(* CODESYS project STAS-60.project

Project tree, tasks and I/O mapping:
  Device : XC303 (Preview), Eaton Automation, version 3.5.11.10
      unmapped channels: Output, Input
    application Application
      libraries: Standard, * (System); CAA CiA 405, 3.5.8.0 (CAA Technical Workgroup); Serial Communication, 3.5.7.0 (3S - Smart Software Solutions GmbH)
      task MainTask (cyclic, interval t#200ms, priority 1) calls PLC_PRG
      task VISU_TASK (cyclic, interval t#200ms, priority 1) calls VisuElems.Visu_Prg
      task TrendRecordingTask (cyclic, interval 100 ms, priority 31) calls VisuTrendStorageAccess.GlobalInstances.g_TrendRecordingManager.CyclicCall
      program PLC_PRG [ST]
      global variables GVL
      visualisation Visualization
    CANbus : CANbus, Eaton Automation, order no. 
      , version 3.5.10.0
      CANopen_Manager : CANopen_Manager, Eaton Automation, order no. 
      , version 3.5.10.0
          settings: ConfigVersion = 50659584
        XNE_GWBR_CANOPEN : XNE-GWBR-CANOPEN, Eaton Automation, order no. 107591, version Revision=16#00040017, FileVersion=4.24
            settings: NODEIDSAVED = 2; SDO Timeout = 1000000; PDO_Autoconfig = TRUE; EXPERTSETTINGS = False; Emergency-General Parameters.Emergency COBID = 16#00000082; Heartbeat-Producer Time = 200; Settings.COBID = 16#00000202; Settings.Transmission Type = 16#FF; Settings.available PDO-Parameter.Inhibit Time available = FALSE; Settings.available PDO-Parameter.Event Timer available = FALSE; Settings.Inhibit Time = 0; Settings.Event Timer = 0; Generic COBID = '$NODEID+16#0200'; Process by CANopenManager = TRUE; Settings.COBID = 16#00000302; Settings.Transmission Type = 16#FF; Settings.available PDO-Parameter.Inhibit Time available = FALSE; Settings.available PDO-Parameter.Event Timer available = FALSE; Settings.Inhibit Time = 0; Settings.Event Timer = 0; Generic COBID = '$NODEID+16#0300'; Process by CANopenManager = TRUE; Settings.COBID = 16#00000282; Settings.Transmission Type = 16#FF; Settings.available PDO-Parameter.Inhibit Time available = TRUE; Settings.available PDO-Parameter.Event Timer available = TRUE; Settings.Inhibit Time = 0; Settings.Event Timer = 0; Generic COBID = '$NODEID+16#0280'; Process by CANopenManager = TRUE; Settings.COBID = 16#00000382; Settings.Transmission Type = 16#FF; Settings.available PDO-Parameter.Inhibit Time available = TRUE; Settings.available PDO-Parameter.Event Timer available = TRUE; Settings.Inhibit Time = 0; Settings.Event Timer = 0; Generic COBID = '$NODEID+16#0380'; Process by CANopenManager = TRUE; Heartbeat-Consuming1.Heartbeat-Time = 300 ms; WriteOutput8Bit : Generic_XN_2DO.Index = 16#6200;
              WriteOutput8Bit : Generic_XN_2DO.Subindex = 16#01; WriteOutput8Bit : Generic_XN_2DO.ObjectLength = 8; WriteOutput8Bit : Generic_XN_2DO_4.Index = 16#6200; WriteOutput8Bit : Generic_XN_2DO_4.Subindex = 16#02; WriteOutput8Bit : Generic_XN_2DO_4.ObjectLength = 8; WriteAnalogueOutput16 : Generic_XNE_4AO.Index = 16#6411; WriteAnalogueOutput16 : Generic_XNE_4AO.Subindex = 16#01; WriteAnalogueOutput16 : Generic_XNE_4AO.ObjectLength = 16; WriteAnalogueOutput16 : Generic_XNE_4AO.Index = 16#6411; WriteAnalogueOutput16 : Generic_XNE_4AO.Subindex = 16#02; WriteAnalogueOutput16 : Generic_XNE_4AO.ObjectLength = 16; WriteAnalogueOutput16 : Generic_XNE_4AO.Index = 16#6411; WriteAnalogueOutput16 : Generic_XNE_4AO.Subindex = 16#03; WriteAnalogueOutput16 : Generic_XNE_4AO.ObjectLength = 16; WriteAnalogueOutput16 : Generic_XNE_4AO.Index = 16#6411; WriteAnalogueOutput16 : Generic_XNE_4AO.Subindex = 16#04; WriteAnalogueOutput16 : Generic_XNE_4AO.ObjectLength = 16; ReadAnalogueInput16Bit : Generic_XNE_8AI.Index = 16#6401; ReadAnalogueInput16Bit : Generic_XNE_8AI.Subindex = 16#01; ReadAnalogueInput16Bit : Generic_XNE_8AI.ObjectLength = 16; ReadAnalogueInput16Bit : Generic_XNE_8AI.Index = 16#6401; ReadAnalogueInput16Bit : Generic_XNE_8AI.Subindex = 16#02; ReadAnalogueInput16Bit : Generic_XNE_8AI.ObjectLength = 16; ReadAnalogueInput16Bit : Generic_XNE_8AI.Index = 16#6401; ReadAnalogueInput16Bit : Generic_XNE_8AI.Subindex = 16#03; ReadAnalogueInput16Bit : Generic_XNE_8AI.ObjectLength = 16; ReadAnalogueInput16Bit : Generic_XNE_8AI.Index = 16#6401; ReadAnalogueInput16Bit : Generic_XNE_8AI.Subindex = 16#04; ReadAnalogueInput16Bit : Generic_XNE_8AI.ObjectLength = 16; ReadAnalogueInput16Bit : Generic_XNE_8AI.Index = 16#6401; ReadAnalogueInput16Bit : Generic_XNE_8AI.Subindex = 16#05; ReadAnalogueInput16Bit : Generic_XNE_8AI.ObjectLength = 16; ReadAnalogueInput16Bit : Generic_XNE_8AI.Index = 16#6401; ReadAnalogueInput16Bit : Generic_XNE_8AI.Subindex = 16#06; ReadAnalogueInput16Bit : Generic_XNE_8AI.ObjectLength = 16; ReadAnalogueInput16Bit : Generic_XNE_8AI.Index = 16#6401; ReadAnalogueInput16Bit : Generic_XNE_8AI.Subindex = 16#07; ReadAnalogueInput16Bit : Generic_XNE_8AI.ObjectLength = 16; ReadAnalogueInput16Bit : Generic_XNE_8AI.Index = 16#6401; ReadAnalogueInput16Bit : Generic_XNE_8AI.Subindex = 16#08;
              ReadAnalogueInput16Bit : Generic_XNE_8AI.ObjectLength = 16; SDO List.Set Guardtime.Index = 16#100C; SDO List.Set Guardtime.Subindex = 16#00; SDO List.Set Guardtime.Value = 16#00000000; SDO List.Set Guardtime.Size = 16; SDO List.Set Guardtime.AbortIfError = FALSE; SDO List.Set Guardtime.JumpToLine = FALSE; SDO List.Set Guardtime.Line = 0; SDO List.Set Lifetime.Index = 16#100D; SDO List.Set Lifetime.Subindex = 16#00; SDO List.Set Lifetime.Value = 16#00000000; SDO List.Set Lifetime.Size = 8; SDO List.Set Lifetime.AbortIfError = FALSE; SDO List.Set Lifetime.JumpToLine = FALSE; SDO List.Set Lifetime.Line = 0; SDO List.Disable Emcy CobID.Index = 16#1014; SDO List.Disable Emcy CobID.Subindex = 16#00; SDO List.Disable Emcy CobID.Value = 16#80000082; SDO List.Disable Emcy CobID.Size = 32; SDO List.Disable Emcy CobID.AbortIfError = FALSE; SDO List.Disable Emcy CobID.JumpToLine = FALSE; SDO List.Disable Emcy CobID.Line = 0; SDO List.Set Emcy CobID.Index = 16#1014; SDO List.Set Emcy CobID.Subindex = 16#00; SDO List.Set Emcy CobID.Value = 16#00000082; SDO List.Set Emcy CobID.Size = 32; SDO List.Set Emcy CobID.AbortIfError = FALSE; SDO List.Set Emcy CobID.JumpToLine = FALSE; SDO List.Set Emcy CobID.Line = 0; SDO List.Set Heartbeat Consumer.Index = 16#1016; SDO List.Set Heartbeat Consumer.Subindex = 16#01; SDO List.Set Heartbeat Consumer.Value = 16#0001012C; SDO List.Set Heartbeat Consumer.Size = 32; SDO List.Set Heartbeat Consumer.AbortIfError = FALSE; SDO List.Set Heartbeat Consumer.JumpToLine = FALSE; SDO List.Set Heartbeat Consumer.Line = 0; SDO List.Set Heartbeat Producer.Index = 16#1017; SDO List.Set Heartbeat Producer.Subindex = 16#00; SDO List.Set Heartbeat Producer.Value = 16#000000C8; SDO List.Set Heartbeat Producer.Size = 16;
              SDO List.Set Heartbeat Producer.AbortIfError = FALSE; SDO List.Set Heartbeat Producer.JumpToLine = FALSE; SDO List.Set Heartbeat Producer.Line = 0; SDO List.Disable PDO.Index = 16#1400; SDO List.Disable PDO.Subindex = 16#01; SDO List.Disable PDO.Value = 16#80000202; SDO List.Disable PDO.Size = 32; SDO List.Disable PDO.AbortIfError = FALSE; SDO List.Disable PDO.JumpToLine = FALSE; SDO List.Disable PDO.Line = 0; SDO List.Set transmission type.Index = 16#1400; SDO List.Set transmission type.Subindex = 16#02; SDO List.Set transmission type.Value = 16#FF; SDO List.Set transmission type.Size = 8; SDO List.Set transmission type.AbortIfError = FALSE; SDO List.Set transmission type.JumpToLine = FALSE; SDO List.Set transmission type.Line = 0; SDO List.Clear pdo mapping.Index = 16#1600; SDO List.Clear pdo mapping.Subindex = 16#00; SDO List.Clear pdo mapping.Value = 16#0; SDO List.Clear pdo mapping.Size = 8; SDO List.Clear pdo mapping.AbortIfError = FALSE; SDO List.Clear pdo mapping.JumpToLine = FALSE; SDO List.Clear pdo mapping.Line = 0; SDO List.Set Mapping.Index = 16#1600; SDO List.Set Mapping.Subindex = 16#01; SDO List.Set Mapping.Value = 16#62000108; SDO List.Set Mapping.Size = 32; SDO List.Set Mapping.AbortIfError = FALSE; SDO List.Set Mapping.JumpToLine = FALSE; SDO List.Set Mapping.Line = 0; SDO List.Set Mapping.Index = 16#1600; SDO List.Set Mapping.Subindex = 16#02; SDO List.Set Mapping.Value = 16#62000208; SDO List.Set Mapping.Size = 32; SDO List.Set Mapping.AbortIfError = FALSE; SDO List.Set Mapping.JumpToLine = FALSE; SDO List.Set Mapping.Line = 0; SDO List.Set number of mappings.Index = 16#1600; SDO List.Set number of mappings.Subindex = 16#00;
              SDO List.Set number of mappings.Value = 16#02; SDO List.Set number of mappings.Size = 8; SDO List.Set number of mappings.AbortIfError = FALSE; SDO List.Set number of mappings.JumpToLine = FALSE; SDO List.Set number of mappings.Line = 0; SDO List.Set and enable COB-ID.Index = 16#1400; SDO List.Set and enable COB-ID.Subindex = 16#01; SDO List.Set and enable COB-ID.Value = 16#00000202; SDO List.Set and enable COB-ID.Size = 32; SDO List.Set and enable COB-ID.AbortIfError = FALSE; SDO List.Set and enable COB-ID.JumpToLine = FALSE; SDO List.Set and enable COB-ID.Line = 0; SDO List.Disable PDO.Index = 16#1401; SDO List.Disable PDO.Subindex = 16#01; SDO List.Disable PDO.Value = 16#80000302; SDO List.Disable PDO.Size = 32; SDO List.Disable PDO.AbortIfError = FALSE; SDO List.Disable PDO.JumpToLine = FALSE; SDO List.Disable PDO.Line = 0; SDO List.Set transmission type.Index = 16#1401; SDO List.Set transmission type.Subindex = 16#02; SDO List.Set transmission type.Value = 16#FF; SDO List.Set transmission type.Size = 8; SDO List.Set transmission type.AbortIfError = FALSE; SDO List.Set transmission type.JumpToLine = FALSE; SDO List.Set transmission type.Line = 0; SDO List.Clear pdo mapping.Index = 16#1601; SDO List.Clear pdo mapping.Subindex = 16#00; SDO List.Clear pdo mapping.Value = 16#0; SDO List.Clear pdo mapping.Size = 8; SDO List.Clear pdo mapping.AbortIfError = FALSE; SDO List.Clear pdo mapping.JumpToLine = FALSE; SDO List.Clear pdo mapping.Line = 0; SDO List.Set Mapping.Index = 16#1601; SDO List.Set Mapping.Subindex = 16#01; SDO List.Set Mapping.Value = 16#64110110; SDO List.Set Mapping.Size = 32; SDO List.Set Mapping.AbortIfError = FALSE; SDO List.Set Mapping.JumpToLine = FALSE; SDO List.Set Mapping.Line = 0;
              SDO List.Set Mapping.Index = 16#1601; SDO List.Set Mapping.Subindex = 16#02; SDO List.Set Mapping.Value = 16#64110210; SDO List.Set Mapping.Size = 32; SDO List.Set Mapping.AbortIfError = FALSE; SDO List.Set Mapping.JumpToLine = FALSE; SDO List.Set Mapping.Line = 0; SDO List.Set Mapping.Index = 16#1601; SDO List.Set Mapping.Subindex = 16#03; SDO List.Set Mapping.Value = 16#64110310; SDO List.Set Mapping.Size = 32; SDO List.Set Mapping.AbortIfError = FALSE; SDO List.Set Mapping.JumpToLine = FALSE; SDO List.Set Mapping.Line = 0; SDO List.Set Mapping.Index = 16#1601; SDO List.Set Mapping.Subindex = 16#04; SDO List.Set Mapping.Value = 16#64110410; SDO List.Set Mapping.Size = 32; SDO List.Set Mapping.AbortIfError = FALSE; SDO List.Set Mapping.JumpToLine = FALSE; SDO List.Set Mapping.Line = 0; SDO List.Set number of mappings.Index = 16#1601; SDO List.Set number of mappings.Subindex = 16#00; SDO List.Set number of mappings.Value = 16#04; SDO List.Set number of mappings.Size = 8; SDO List.Set number of mappings.AbortIfError = FALSE; SDO List.Set number of mappings.JumpToLine = FALSE; SDO List.Set number of mappings.Line = 0; SDO List.Set and enable COB-ID.Index = 16#1401; SDO List.Set and enable COB-ID.Subindex = 16#01; SDO List.Set and enable COB-ID.Value = 16#00000302; SDO List.Set and enable COB-ID.Size = 32; SDO List.Set and enable COB-ID.AbortIfError = FALSE; SDO List.Set and enable COB-ID.JumpToLine = FALSE; SDO List.Set and enable COB-ID.Line = 0; SDO List.Disable PDO.Index = 16#1801; SDO List.Disable PDO.Subindex = 16#01; SDO List.Disable PDO.Value = 16#80000282; SDO List.Disable PDO.Size = 32; SDO List.Disable PDO.AbortIfError = FALSE;
              SDO List.Disable PDO.JumpToLine = FALSE; SDO List.Disable PDO.Line = 0; SDO List.Set transmission type.Index = 16#1801; SDO List.Set transmission type.Subindex = 16#02; SDO List.Set transmission type.Value = 16#FF; SDO List.Set transmission type.Size = 8; SDO List.Set transmission type.AbortIfError = FALSE; SDO List.Set transmission type.JumpToLine = FALSE; SDO List.Set transmission type.Line = 0; SDO List.Set inhibit time.Index = 16#1801; SDO List.Set inhibit time.Subindex = 16#03; SDO List.Set inhibit time.Value = 16#0000; SDO List.Set inhibit time.Size = 16; SDO List.Set inhibit time.AbortIfError = FALSE; SDO List.Set inhibit time.JumpToLine = FALSE; SDO List.Set inhibit time.Line = 0; SDO List.Set event time.Index = 16#1801; SDO List.Set event time.Subindex = 16#05; SDO List.Set event time.Value = 16#0000; SDO List.Set event time.Size = 16; SDO List.Set event time.AbortIfError = FALSE; SDO List.Set event time.JumpToLine = FALSE; SDO List.Set event time.Line = 0; SDO List.Clear pdo mapping.Index = 16#1A01; SDO List.Clear pdo mapping.Subindex = 16#00; SDO List.Clear pdo mapping.Value = 16#0; SDO List.Clear pdo mapping.Size = 8; SDO List.Clear pdo mapping.AbortIfError = FALSE; SDO List.Clear pdo mapping.JumpToLine = FALSE; SDO List.Clear pdo mapping.Line = 0; SDO List.Set Mapping.Index = 16#1A01; SDO List.Set Mapping.Subindex = 16#01; SDO List.Set Mapping.Value = 16#64010110; SDO List.Set Mapping.Size = 32; SDO List.Set Mapping.AbortIfError = FALSE; SDO List.Set Mapping.JumpToLine = FALSE; SDO List.Set Mapping.Line = 0; SDO List.Set Mapping.Index = 16#1A01; SDO List.Set Mapping.Subindex = 16#02; SDO List.Set Mapping.Value = 16#64010210;
              SDO List.Set Mapping.Size = 32; SDO List.Set Mapping.AbortIfError = FALSE; SDO List.Set Mapping.JumpToLine = FALSE; SDO List.Set Mapping.Line = 0; SDO List.Set Mapping.Index = 16#1A01; SDO List.Set Mapping.Subindex = 16#03; SDO List.Set Mapping.Value = 16#64010310; SDO List.Set Mapping.Size = 32; SDO List.Set Mapping.AbortIfError = FALSE; SDO List.Set Mapping.JumpToLine = FALSE; SDO List.Set Mapping.Line = 0; SDO List.Set Mapping.Index = 16#1A01; SDO List.Set Mapping.Subindex = 16#04; SDO List.Set Mapping.Value = 16#64010410; SDO List.Set Mapping.Size = 32; SDO List.Set Mapping.AbortIfError = FALSE; SDO List.Set Mapping.JumpToLine = FALSE; SDO List.Set Mapping.Line = 0; SDO List.Set number of mappings.Index = 16#1A01; SDO List.Set number of mappings.Subindex = 16#00; SDO List.Set number of mappings.Value = 16#04; SDO List.Set number of mappings.Size = 8; SDO List.Set number of mappings.AbortIfError = FALSE; SDO List.Set number of mappings.JumpToLine = FALSE; SDO List.Set number of mappings.Line = 0; SDO List.Set and enable COB-ID.Index = 16#1801; SDO List.Set and enable COB-ID.Subindex = 16#01; SDO List.Set and enable COB-ID.Value = 16#00000282; SDO List.Set and enable COB-ID.Size = 32; SDO List.Set and enable COB-ID.AbortIfError = FALSE; SDO List.Set and enable COB-ID.JumpToLine = FALSE; SDO List.Set and enable COB-ID.Line = 0; SDO List.Disable PDO.Index = 16#1802; SDO List.Disable PDO.Subindex = 16#01; SDO List.Disable PDO.Value = 16#80000382; SDO List.Disable PDO.Size = 32; SDO List.Disable PDO.AbortIfError = FALSE; SDO List.Disable PDO.JumpToLine = FALSE; SDO List.Disable PDO.Line = 0; SDO List.Set transmission type.Index = 16#1802;
              SDO List.Set transmission type.Subindex = 16#02; SDO List.Set transmission type.Value = 16#FF; SDO List.Set transmission type.Size = 8; SDO List.Set transmission type.AbortIfError = FALSE; SDO List.Set transmission type.JumpToLine = FALSE; SDO List.Set transmission type.Line = 0; SDO List.Set inhibit time.Index = 16#1802; SDO List.Set inhibit time.Subindex = 16#03; SDO List.Set inhibit time.Value = 16#0000; SDO List.Set inhibit time.Size = 16; SDO List.Set inhibit time.AbortIfError = FALSE; SDO List.Set inhibit time.JumpToLine = FALSE; SDO List.Set inhibit time.Line = 0; SDO List.Set event time.Index = 16#1802; SDO List.Set event time.Subindex = 16#05; SDO List.Set event time.Value = 16#0000; SDO List.Set event time.Size = 16; SDO List.Set event time.AbortIfError = FALSE; SDO List.Set event time.JumpToLine = FALSE; SDO List.Set event time.Line = 0; SDO List.Clear pdo mapping.Index = 16#1A02; SDO List.Clear pdo mapping.Subindex = 16#00; SDO List.Clear pdo mapping.Value = 16#0; SDO List.Clear pdo mapping.Size = 8; SDO List.Clear pdo mapping.AbortIfError = FALSE; SDO List.Clear pdo mapping.JumpToLine = FALSE; SDO List.Clear pdo mapping.Line = 0; SDO List.Set Mapping.Index = 16#1A02; SDO List.Set Mapping.Subindex = 16#01; SDO List.Set Mapping.Value = 16#64010510; SDO List.Set Mapping.Size = 32; SDO List.Set Mapping.AbortIfError = FALSE; SDO List.Set Mapping.JumpToLine = FALSE; SDO List.Set Mapping.Line = 0; SDO List.Set Mapping.Index = 16#1A02; SDO List.Set Mapping.Subindex = 16#02; SDO List.Set Mapping.Value = 16#64010610; SDO List.Set Mapping.Size = 32; SDO List.Set Mapping.AbortIfError = FALSE; SDO List.Set Mapping.JumpToLine = FALSE;
              SDO List.Set Mapping.Line = 0; SDO List.Set Mapping.Index = 16#1A02; SDO List.Set Mapping.Subindex = 16#03; SDO List.Set Mapping.Value = 16#64010710; SDO List.Set Mapping.Size = 32; SDO List.Set Mapping.AbortIfError = FALSE; SDO List.Set Mapping.JumpToLine = FALSE; SDO List.Set Mapping.Line = 0; SDO List.Set Mapping.Index = 16#1A02; SDO List.Set Mapping.Subindex = 16#04; SDO List.Set Mapping.Value = 16#64010810; SDO List.Set Mapping.Size = 32; SDO List.Set Mapping.AbortIfError = FALSE; SDO List.Set Mapping.JumpToLine = FALSE; SDO List.Set Mapping.Line = 0; SDO List.Set number of mappings.Index = 16#1A02; SDO List.Set number of mappings.Subindex = 16#00; SDO List.Set number of mappings.Value = 16#04; SDO List.Set number of mappings.Size = 8; SDO List.Set number of mappings.AbortIfError = FALSE; SDO List.Set number of mappings.JumpToLine = FALSE; SDO List.Set number of mappings.Line = 0; SDO List.Set and enable COB-ID.Index = 16#1802; SDO List.Set and enable COB-ID.Subindex = 16#01; SDO List.Set and enable COB-ID.Value = 16#00000382; SDO List.Set and enable COB-ID.Size = 32; SDO List.Set and enable COB-ID.AbortIfError = FALSE; SDO List.Set and enable COB-ID.JumpToLine = FALSE; SDO List.Set and enable COB-ID.Line = 0; ConfigVersion = 50659584
          Generic_XN_2DO : Generic XN-2DO, Eaton Automation, order no. 0, version Revision=16#00040017, FileVersion=4.24
              settings: Number of Params = 1; WriteOutput8Bit : Generic_XN_2DO.Index = 16#6200; WriteOutput8Bit : Generic_XN_2DO.Subindex = 16#01; WriteOutput8Bit : Generic_XN_2DO.Startbit = 0; WriteOutput8Bit : Generic_XN_2DO.Endbit = 1
              unmapped channels: WriteOutput8Bit : Generic_XN_2DO
          Generic_XN_2DO_1 : Generic XN-2DO, Eaton Automation, order no. 0, version Revision=16#00040017, FileVersion=4.24
              settings: Number of Params = 1; WriteOutput8Bit : Generic_XN_2DO.Index = 16#6200; WriteOutput8Bit : Generic_XN_2DO.Subindex = 16#01; WriteOutput8Bit : Generic_XN_2DO.Startbit = 2; WriteOutput8Bit : Generic_XN_2DO.Endbit = 3
              unmapped channels: WriteOutput8Bit : Generic_XN_2DO
          Generic_XN_2DO_2 : Generic XN-2DO, Eaton Automation, order no. 0, version Revision=16#00040017, FileVersion=4.24
              settings: Number of Params = 1; WriteOutput8Bit : Generic_XN_2DO.Index = 16#6200; WriteOutput8Bit : Generic_XN_2DO.Subindex = 16#01; WriteOutput8Bit : Generic_XN_2DO.Startbit = 4; WriteOutput8Bit : Generic_XN_2DO.Endbit = 5
              unmapped channels: WriteOutput8Bit : Generic_XN_2DO
          Generic_XN_2DO_3 : Generic XN-2DO, Eaton Automation, order no. 0, version Revision=16#00040017, FileVersion=4.24
              settings: Number of Params = 1; WriteOutput8Bit : Generic_XN_2DO.Index = 16#6200; WriteOutput8Bit : Generic_XN_2DO.Subindex = 16#01; WriteOutput8Bit : Generic_XN_2DO.Startbit = 6; WriteOutput8Bit : Generic_XN_2DO.Endbit = 7
              unmapped channels: WriteOutput8Bit : Generic_XN_2DO
          Generic_XN_2DO_4 : Generic XN-2DO, Eaton Automation, order no. 0, version Revision=16#00040017, FileVersion=4.24
              settings: Number of Params = 1; WriteOutput8Bit : Generic_XN_2DO_4.Index = 16#6200; WriteOutput8Bit : Generic_XN_2DO_4.Subindex = 16#02; WriteOutput8Bit : Generic_XN_2DO_4.Startbit = 0; WriteOutput8Bit : Generic_XN_2DO_4.Endbit = 1
              unmapped channels: WriteOutput8Bit : Generic_XN_2DO_4
          Generic_XN_2DO_5 : Generic XN-2DO, Eaton Automation, order no. 0, version Revision=16#00040017, FileVersion=4.24
              settings: Number of Params = 1; WriteOutput8Bit : Generic_XN_2DO_4.Index = 16#6200; WriteOutput8Bit : Generic_XN_2DO_4.Subindex = 16#02; WriteOutput8Bit : Generic_XN_2DO_4.Startbit = 2; WriteOutput8Bit : Generic_XN_2DO_4.Endbit = 3
              unmapped channels: WriteOutput8Bit : Generic_XN_2DO_4
          Generic_XN_2DO_6 : Generic XN-2DO, Eaton Automation, order no. 0, version Revision=16#00040017, FileVersion=4.24
              settings: Number of Params = 1; WriteOutput8Bit : Generic_XN_2DO_4.Index = 16#6200; WriteOutput8Bit : Generic_XN_2DO_4.Subindex = 16#02; WriteOutput8Bit : Generic_XN_2DO_4.Startbit = 4; WriteOutput8Bit : Generic_XN_2DO_4.Endbit = 5
              unmapped channels: WriteOutput8Bit : Generic_XN_2DO_4
          Generic_XN_2DO_7 : Generic XN-2DO, Eaton Automation, order no. 0, version Revision=16#00040017, FileVersion=4.24
              settings: Number of Params = 1; WriteOutput8Bit : Generic_XN_2DO_4.Index = 16#6200; WriteOutput8Bit : Generic_XN_2DO_4.Subindex = 16#02; WriteOutput8Bit : Generic_XN_2DO_4.Startbit = 6; WriteOutput8Bit : Generic_XN_2DO_4.Endbit = 7
              unmapped channels: WriteOutput8Bit : Generic_XN_2DO_4
          Generic_XNE_4AO : Generic XNE-4AO, Eaton Automation, order no. 0, version Revision=16#00040017, FileVersion=4.24
              settings: Number of Params = 4; WriteAnalogueOutput16 : Generic_XNE_4AO.Index = 16#6411; WriteAnalogueOutput16 : Generic_XNE_4AO.Subindex = 16#01; WriteAnalogueOutput16 : Generic_XNE_4AO.Startbit = 0; WriteAnalogueOutput16 : Generic_XNE_4AO.Endbit = 15; WriteAnalogueOutput16 : Generic_XNE_4AO.Index = 16#6411; WriteAnalogueOutput16 : Generic_XNE_4AO.Subindex = 16#02; WriteAnalogueOutput16 : Generic_XNE_4AO.Startbit = 0; WriteAnalogueOutput16 : Generic_XNE_4AO.Endbit = 15; WriteAnalogueOutput16 : Generic_XNE_4AO.Index = 16#6411; WriteAnalogueOutput16 : Generic_XNE_4AO.Subindex = 16#03; WriteAnalogueOutput16 : Generic_XNE_4AO.Startbit = 0; WriteAnalogueOutput16 : Generic_XNE_4AO.Endbit = 15; WriteAnalogueOutput16 : Generic_XNE_4AO.Index = 16#6411; WriteAnalogueOutput16 : Generic_XNE_4AO.Subindex = 16#04; WriteAnalogueOutput16 : Generic_XNE_4AO.Startbit = 0; WriteAnalogueOutput16 : Generic_XNE_4AO.Endbit = 15
              unmapped channels: WriteAnalogueOutput16 : Generic_XNE_4AO, WriteAnalogueOutput16 : Generic_XNE_4AO, WriteAnalogueOutput16 : Generic_XNE_4AO, WriteAnalogueOutput16 : Generic_XNE_4AO
          Generic_XNE_8AI : Generic XNE-8AI, Eaton Automation, order no. 0, version Revision=16#00040017, FileVersion=4.24
              settings: Number of Params = 8; ReadAnalogueInput16Bit : Generic_XNE_8AI.Index = 16#6401; ReadAnalogueInput16Bit : Generic_XNE_8AI.Subindex = 16#01; ReadAnalogueInput16Bit : Generic_XNE_8AI.Startbit = 0; ReadAnalogueInput16Bit : Generic_XNE_8AI.Endbit = 15; ReadAnalogueInput16Bit : Generic_XNE_8AI.Index = 16#6401; ReadAnalogueInput16Bit : Generic_XNE_8AI.Subindex = 16#02; ReadAnalogueInput16Bit : Generic_XNE_8AI.Startbit = 0; ReadAnalogueInput16Bit : Generic_XNE_8AI.Endbit = 15; ReadAnalogueInput16Bit : Generic_XNE_8AI.Index = 16#6401; ReadAnalogueInput16Bit : Generic_XNE_8AI.Subindex = 16#03; ReadAnalogueInput16Bit : Generic_XNE_8AI.Startbit = 0; ReadAnalogueInput16Bit : Generic_XNE_8AI.Endbit = 15; ReadAnalogueInput16Bit : Generic_XNE_8AI.Index = 16#6401; ReadAnalogueInput16Bit : Generic_XNE_8AI.Subindex = 16#04; ReadAnalogueInput16Bit : Generic_XNE_8AI.Startbit = 0; ReadAnalogueInput16Bit : Generic_XNE_8AI.Endbit = 15; ReadAnalogueInput16Bit : Generic_XNE_8AI.Index = 16#6401; ReadAnalogueInput16Bit : Generic_XNE_8AI.Subindex = 16#05; ReadAnalogueInput16Bit : Generic_XNE_8AI.Startbit = 0; ReadAnalogueInput16Bit : Generic_XNE_8AI.Endbit = 15; ReadAnalogueInput16Bit : Generic_XNE_8AI.Index = 16#6401; ReadAnalogueInput16Bit : Generic_XNE_8AI.Subindex = 16#06; ReadAnalogueInput16Bit : Generic_XNE_8AI.Startbit = 0; ReadAnalogueInput16Bit : Generic_XNE_8AI.Endbit = 15; ReadAnalogueInput16Bit : Generic_XNE_8AI.Index = 16#6401; ReadAnalogueInput16Bit : Generic_XNE_8AI.Subindex = 16#07; ReadAnalogueInput16Bit : Generic_XNE_8AI.Startbit = 0; ReadAnalogueInput16Bit : Generic_XNE_8AI.Endbit = 15; ReadAnalogueInput16Bit : Generic_XNE_8AI.Index = 16#6401; ReadAnalogueInput16Bit : Generic_XNE_8AI.Subindex = 16#08; ReadAnalogueInput16Bit : Generic_XNE_8AI.Startbit = 0; ReadAnalogueInput16Bit : Generic_XNE_8AI.Endbit = 15
              unmapped channels: ReadAnalogueInput16Bit : Generic_XNE_8AI, ReadAnalogueInput16Bit : Generic_XNE_8AI, ReadAnalogueInput16Bit : Generic_XNE_8AI, ReadAnalogueInput16Bit : Generic_XNE_8AI, ReadAnalogueInput16Bit : Generic_XNE_8AI, ReadAnalogueInput16Bit : Generic_XNE_8AI, ReadAnalogueInput16Bit : Generic_XNE_8AI, ReadAnalogueInput16Bit : Generic_XNE_8AI
    Ethernet : Ethernet, Eaton Automation, version 3.5.11.0
      ModbusTCP_Slave_Device : ModbusTCP Slave Device, 3S - Smart Software Solutions GmbH, version 3.5.11.0
          unmapped channels: Входы, Выходы
  libraries: VisuSymbols, 3.5.10.0 (System)
  text list GlobalTextList
*)

// Device/Application/GVL
{attribute 'qualified_only'}
VAR_GLOBAL
	
	hiPres AT %IW2: WORD; (*Датчик высокго давления на гидроразпределителе*)
	lowPres AT %IW4: WORD; (*Датчик низкого давления на гидроразпределителе*)
	mowAbsorb AT %IW6: WORD; (*Датчик хода гидроамортизатора*)
	compressPress AT %IW8: WORD; (*Датчик давления на сжатие*)
	decomressPress AT %IW10: WORD; (*Датчик давления на росжатие*)
	
	temperatuteOil : WORD; (*Датчик температуры масла*)
	levelOil : WORD; (*Датчик уровня масла*)
	
	defectHiPresSens: BOOL; (*Неисправность датчика высокго давления на гидроразпределителе*)
	defectLowPresSens: BOOL; (*Неисправность датчика низкого давления на гидроразпределителе*)
	defectMowAbsorbSens: BOOL; (*Неисправность датчика хода гидроамортизатора*)
	defectDecomressPressSens: BOOL; (*Неисправность датчика давления на росжатие*)
	defectCompressPressSens: BOOL; (*Неисправность датчика давления на сжатие*)
	defectTemperatuteOilSens: BOOL; (*Неисправность датчика температуры масла*)
	defectLevelOilSens: BOOL; (*Неисправность датчика уровня масла*)
		
	SOL1 : BOOL; (* Соленоид высокого давления *)
	SOL2 : BOOL; (* Соленоид низкого давления *)
	SOL3: BOOL; (* Соленоид растяжения *)
	SOL4: BOOL; (* Соленоид сжатия *)
	SOL5: BOOL; (* Соленоид без давления *)
	
	SOL10: BOOL; (* Соленоид перепад давления Сжатие *)
	SOL11: BOOL; (* Соленоид перепад давления Растяжение *)
	
	pumpOn: BOOL; (*Включение насоса*)
	pumpStart: BOOL; (*Разгон насоса*)
	pumpWork: BOOL; (*Рабочий режим насоса*)
	
	timePumpStart: TIME; (*Время разгона насоса*)
	
	heaterOil: BOOL; (*Подогрева масла*)
	coolerOil: BOOL; (*Охлаждение масла*)
	
	
	normalLoadMode: BOOL; (*Режим нормальной нагрузки*)
	openMode: BOOL;  (*Проверка открытия клапана*)
	resistanceMode: BOOL; (*Режим испытания сопротивления ГА без нагрузки (холостой ход)*)
	speedCloseMode: BOOL; (*Скорость закрытия*)
	
	nProcess: INT;
	kokoetoChislo: WORD;

END_VAR

// Device/Application/PLC_PRG
PROGRAM PLC_PRG
VAR

	hiPres : WORD:=10; (*Датчик высокго давления на гидроразпределителе*)
	lowPres : WORD:=10; (*Датчик низкого давления на гидроразпределителе*)
	mowAbsorb : WORD:=10; (*Датчик хода гидроамортизатора*)
	compressPress : WORD:=10; (*Датчик давления на сжатие*)
	decomressPress : WORD:=10; (*Датчик давления на росжатие*)
	
	temperatuteOil : WORD:=10; (*Датчик температуры масла*)
	levelOil : WORD:=10; (*Датчик уровня масла*)
	
	leftMowAbsorb: WORD;
	rightMowAbsorb: WORD;
	
	TONInst : TON ;
	setSOL10: BOOL;
	
	
	TOFInst : TOF;
	timeSOL10: TIME:=T#5S; 
		
	TONPump : TON ;
	setPump: BOOL;
	timePump: TIME:=T#5S;
	
	TONnormalMode:TON;
	TOFnormalMode:TOF;
	setNormalMode: BOOL;
	timeNormalMode : TIME:=T#10S;
	
	countNormalMode : INT:=1;
	
	tonSOL1 : TON;
	tofSOL1 : TOF;
	
	tonSOL2 : TON;
	tofSOL2 : TOF;
	
	tonSOL3 : TON;
	tofSOL3 : TOF;
	
	tonSOL4 : TON;
	tofSOL4 : TOF;
	
	tonSOL10 : TON;
	tofSOL10 : TOF;
	
	tonSOL11 : TON;
	tofSOL11 : TOF;
	
	onButton:BOOL;
	
END_VAR

(*Проверка работоспособности датчиков. Анализ токовой петли*)

onButton:= NOT(GVL.pumpWork);

(*Датчик высокого давления*)
IF (hiPres<4 OR hiPres>20 )THEN
		GVL.defectHiPresSens := TRUE;
		ELSE
		GVL.defectHiPresSens := FALSE;
END_IF

(*Датчик низкого давления*)
IF (lowPres<4 OR lowPres>20 )THEN
		GVL.defectLowPresSens := TRUE;
		ELSE
		GVL.defectLowPresSens := FALSE;
END_IF

(*Датчик сжатия*)
IF (compressPress<4 OR compressPress>20 )THEN
		GVL.defectCompressPressSens := TRUE;
		ELSE
		GVL.defectCompressPressSens := FALSE;
END_IF

(*Датчик расжатия*)
IF (decomressPress<4 OR decomressPress>20 )THEN
		GVL.defectDecomressPressSens := TRUE;
		ELSE
		GVL.defectDecomressPressSens := FALSE;
END_IF

(*Датчик температуры масла*)
IF (temperatuteOil<4 OR temperatuteOil>20 )THEN
		GVL.defectTemperatuteOilSens := TRUE;
		ELSE
		GVL.defectTemperatuteOilSens := FALSE;
END_IF

(*Датчик хода гидроамортизатора*)
IF (mowAbsorb<4 OR mowAbsorb>20 )THEN
		GVL.defectMowAbsorbSens := TRUE;
		ELSE
		GVL.defectMowAbsorbSens := FALSE;
END_IF
(*-----------------------------------------------------------*)

(*Ржеим нагрева и охлаждения масла*)

(*Охлаждение*)
IF (temperatuteOil>=16 AND temperatuteOil<=20) THEN
	GVL.coolerOil:=TRUE;
ELSE
	GVL.coolerOil:=FALSE;
END_IF

(*Нагрев*)
IF (temperatuteOil>=4 AND temperatuteOil<=8) THEN
	GVL.heaterOil:=TRUE;
	//TONInst(IN:= GVL.heaterOil, PT:= timeSOL10, Q=> GVL.SOL10);
	//TOFInst(IN:= GVL.heaterOil, PT:= timeSOL10);						
ELSE
	GVL.heaterOil:=FALSE;	
	//TOFInst(IN:= GVL.heaterOil, PT:= timeSOL10, Q=> GVL.SOL10);
	//TONInst(IN := GVL.heaterOil, PT:= timeSOL10);
END_IF
(*-----------------------------------------------------------*)

(*РАбота с електро насосом *)
IF (GVL.pumpOn = TRUE) THEN	
	IF (GVL.pumpWork = FALSE)THEN
		GVL.pumpStart := TRUE;
		TONPump(IN:=GVL.pumpStart, PT:= timePump,Q=>GVL.pumpWork );
	END_IF
ELSE
	GVL.pumpStart := FALSE;
	GVL.pumpWork := FALSE;
	TONPump(IN:=GVL.pumpStart, PT:= timePump);
END_IF
(*------------------------------------------------------------*)


(*Режим нормальной нагрузки*)
IF (GVL.normalLoadMode = TRUE AND GVL.pumpOn=TRUE) THEN
	
CASE countNormalMode OF
1:
	GVL.SOL1:=TRUE;
	tonSOL10 (IN:=TRUE,PT:=T#3S, Q=>GVL.SOL10);
	tonSOL3 (IN:=TRUE,PT:=T#5S, Q=>GVL.SOL3);
	TONnormalMode (IN:=TRUE,PT:=T#10S, Q=>GVL.SOL5);
	
	IF (GVL.SOL5=TRUE) THEN
		TONnormalMode (IN:=FALSE,PT:=T#0S);
		TOFnormalMode (IN:=TRUE,PT:=T#0S);
		tonSOL10 (IN:=FALSE,PT:=T#0S);
		tonSOL3 (IN:=FALSE,PT:=T#0S);
		countNormalMode:=2;
	END_IF
2:
	TOFnormalMode (IN:=FALSE,PT:=T#3S, Q=>GVL.SOL5);
	IF (GVL.SOL5=FALSE) THEN
		TOFnormalMode (IN:=TRUE,PT:=T#0S);		
		countNormalMode:=3;
	END_IF

3:
	tofSOL10 (IN:=FALSE,PT:=T#4S, Q=>GVL.SOL10);
	tofSOL3 (IN:=FALSE,PT:=T#2S, Q=>GVL.SOL3);
	IF (GVL.SOL10=FALSE) THEN
		tofSOL10 (IN:=TRUE,PT:=T#0S);
		tofSOL3 (IN:=TRUE,PT:=T#0S);
	countNormalMode:=4;
	END_IF
4:
	tonSOL11 (IN:=TRUE,PT:=T#3S, Q=>GVL.SOL11);
	tonSOL4 (IN:=TRUE,PT:=T#6S, Q=>GVL.SOL4);
	TONnormalMode (IN:=TRUE,PT:=T#10S, Q=>GVL.SOL5);
	IF (GVL.SOL5=TRUE) THEN
		TONnormalMode (IN:=FALSE,PT:=T#0S);
		tonSOL11 (IN:=FALSE,PT:=T#0S);
		tonSOL4 (IN:=FALSE,PT:=T#0S);
		countNormalMode:=5;
	END_IF
	
5:
	TOFnormalMode (IN:=FALSE,PT:=T#2S, Q=>GVL.SOL5);
	IF (GVL.SOL5=FALSE) THEN
		TOFnormalMode (IN:=TRUE,PT:=T#0S);		
		countNormalMode:=6;
	END_IF
	
6:
	tofSOL11 (IN:=FALSE,PT:=T#4S, Q=>GVL.SOL11);
	tofSOL4 (IN:=FALSE,PT:=T#2S, Q=>GVL.SOL4);
	IF (GVL.SOL11=FALSE) THEN
		tofSOL11 (IN:=TRUE,PT:=T#0S);
		tofSOL4 (IN:=TRUE,PT:=T#0S);
	countNormalMode:=7;
	END_IF
ELSE
	
	countNormalMode:=1;
	GVL.normalLoadMode := FALSE;
		GVL.SOL1:=FALSE;
END_CASE;

END_IF
(*-------------------------------------------------------------*)

(*Режим проверки открытия клапанов*)
IF (GVL.openMode = TRUE AND GVL.pumpOn=TRUE) THEN
	CASE countNormalMode OF	
	1:
		GVL.SOL1:=TRUE;
		tonSOL10 (IN:=TRUE,PT:=T#3S, Q=>GVL.SOL10);
		tonSOL3 (IN:=TRUE,PT:=T#5S, Q=>GVL.SOL3);
		TONnormalMode (IN:=TRUE,PT:=T#10S, Q=>GVL.SOL5);
	
		IF (mowAbsorb>=24) THEN
			TONnormalMode (IN:=FALSE,PT:=T#0S);
			TOFnormalMode (IN:=TRUE,PT:=T#0S);
			tonSOL10 (IN:=FALSE,PT:=T#0S);
			tonSOL3 (IN:=FALSE,PT:=T#0S);
			countNormalMode:=2;
		END_IF
	
	2:
		TOFnormalMode (IN:=FALSE,PT:=T#3S, Q=>GVL.SOL5);
		IF (GVL.SOL5=FALSE) THEN
			TOFnormalMode (IN:=TRUE,PT:=T#0S);		
			countNormalMode:=3;
		END_IF
	
	3:
		tofSOL10 (IN:=FALSE,PT:=T#4S, Q=>GVL.SOL10);
		tofSOL3 (IN:=FALSE,PT:=T#2S, Q=>GVL.SOL3);
		IF (GVL.SOL10=FALSE) THEN
		tofSOL10 (IN:=TRUE,PT:=T#0S);
		tofSOL3 (IN:=TRUE,PT:=T#0S);
		countNormalMode:=4;
		END_IF
	
	4:
		tonSOL11 (IN:=TRUE,PT:=T#3S, Q=>GVL.SOL11);
		tonSOL4 (IN:=TRUE,PT:=T#6S, Q=>GVL.SOL4);
		TONnormalMode (IN:=TRUE,PT:=T#10S, Q=>GVL.SOL5);
		IF (mowAbsorb<=14) THEN
		TONnormalMode (IN:=FALSE,PT:=T#0S);
		tonSOL11 (IN:=FALSE,PT:=T#0S);
		tonSOL4 (IN:=FALSE,PT:=T#0S);
		countNormalMode:=5;
		END_IF
	
	5:
		TOFnormalMode (IN:=FALSE,PT:=T#2S, Q=>GVL.SOL5);
		IF (GVL.SOL5=FALSE) THEN
		TOFnormalMode (IN:=TRUE,PT:=T#0S);		
		countNormalMode:=6;
		END_IF
	
	6:
		tofSOL11 (IN:=FALSE,PT:=T#4S, Q=>GVL.SOL11);
		tofSOL4 (IN:=FALSE,PT:=T#2S, Q=>GVL.SOL4);
		IF (GVL.SOL11=FALSE) THEN
		tofSOL11 (IN:=TRUE,PT:=T#0S);
		tofSOL4 (IN:=TRUE,PT:=T#0S);
		countNormalMode:=7;
		END_IF
	
	ELSE
		countNormalMode:=1;
		GVL.openMode := FALSE;
		GVL.SOL1:=FALSE;
	END_CASE
END_IF
(*-------------------------------------------------------------*)

(*Испытание на сопротивление ГА без нагрузки*)
IF (GVL.resistanceMode = TRUE AND GVL.pumpOn=TRUE) THEN
	
CASE countNormalMode OF
	1:
		GVL.SOL2:=TRUE;
		//tonSOL10 (IN:=TRUE,PT:=T#3S, Q=>GVL.SOL10);
		tonSOL3 (IN:=TRUE,PT:=T#5S, Q=>GVL.SOL3);
		TONnormalMode (IN:=TRUE,PT:=T#10S, Q=>GVL.SOL5);
				
		IF (mowAbsorb>=29) THEN
			TONnormalMode (IN:=FALSE,PT:=T#0S);
			TOFnormalMode (IN:=TRUE,PT:=T#0S);
			//tonSOL10 (IN:=FALSE,PT:=T#0S);
			tonSOL3 (IN:=FALSE,PT:=T#0S);
			countNormalMode:=2;
		END_IF
	2:
		TOFnormalMode (IN:=FALSE,PT:=T#3S, Q=>GVL.SOL5);
		IF (GVL.SOL5=FALSE) THEN
			TOFnormalMode (IN:=TRUE,PT:=T#0S);		
			countNormalMode:=3;
		END_IF
		
	3:
		//tofSOL10 (IN:=FALSE,PT:=T#4S, Q=>GVL.SOL10);
		tofSOL3 (IN:=FALSE,PT:=T#2S, Q=>GVL.SOL3);
		IF (GVL.SOL3=FALSE) THEN
		//tofSOL10 (IN:=TRUE,PT:=T#0S);
		tofSOL3 (IN:=TRUE,PT:=T#0S);
		countNormalMode:=4;
		END_IF
	
	4:
		//tonSOL11 (IN:=TRUE,PT:=T#3S, Q=>GVL.SOL11);
		tonSOL4 (IN:=TRUE,PT:=T#6S, Q=>GVL.SOL4);
		TONnormalMode (IN:=TRUE,PT:=T#10S, Q=>GVL.SOL5);
		IF (mowAbsorb<=9) THEN
		TONnormalMode (IN:=FALSE,PT:=T#0S);
		//tonSOL11 (IN:=FALSE,PT:=T#0S);
		tonSOL4 (IN:=FALSE,PT:=T#0S);
		countNormalMode:=5;
		END_IF
	
	5:
		TOFnormalMode (IN:=FALSE,PT:=T#2S, Q=>GVL.SOL5);
		IF (GVL.SOL5=FALSE) THEN
		TOFnormalMode (IN:=TRUE,PT:=T#0S);		
		countNormalMode:=6;
		END_IF
		
	6:
		//tofSOL11 (IN:=FALSE,PT:=T#4S, Q=>GVL.SOL11);
		tofSOL4 (IN:=FALSE,PT:=T#2S, Q=>GVL.SOL4);
		IF (GVL.SOL4=FALSE) THEN
		//tofSOL11 (IN:=TRUE,PT:=T#0S);
		tofSOL4 (IN:=TRUE,PT:=T#0S);
		countNormalMode:=7;
		END_IF
		
	ELSE
		countNormalMode:=1;
		GVL.resistanceMode := FALSE;
		GVL.SOL2:=FALSE;
	
END_CASE

END_IF
(*-------------------------------------------------------------*)

(*Испытание скорости закрытия клапанов ГА*)
(*-------------------------------------------------------------*)

IF (mowAbsorb>=19 AND mowAbsorb<34) THEN	
rightMowAbsorb:=mowAbsorb-19;
END_IF

IF (mowAbsorb>4 AND mowAbsorb<=19) THEN	
leftMowAbsorb:=19-mowAbsorb;
END_IF

END_PROGRAM

// Device/Application/Visualization
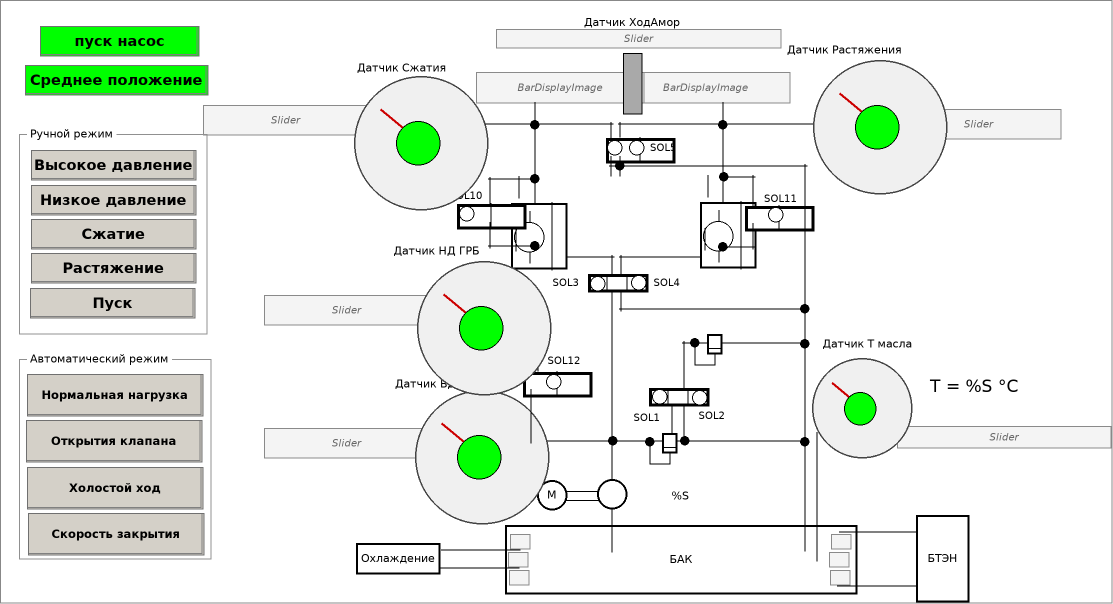
VISUALIZATION Visualization  // 1113x604
VAR_IN_OUT
END_VAR
VAR
	bResetTrigger : BOOL;
	bStop : BOOL;
	bStore : BOOL;
	sStoreFilename : STRING;
	bRestore : BOOL;
	sRestoreFilename : STRING;
END_VAR
    Rectangle (505,525 352x69), "БАК"
    Line (684,443) (684,341), colour toggle: GVL.SOL2
    Line (805,441) (505,441), colour toggle: GVL.pumpWork
    Line (805,343) (682,343), colour toggle: GVL.SOL2
    Slider (897,426 214x22), variable: PLC_PRG.temperatuteOil, scale 0..24
    Rectangle (927,371 95x30), "T = %S °C", text variable: PLC_PRG.temperatuteOil
    Slider (264,428 165x30), variable: PLC_PRG.hiPres, scale 0..25
    Slider (264,295 165x30), variable: PLC_PRG.lowPres, scale 0..25
    Slider (203,105 165x30), variable: PLC_PRG.compressPress, scale 0..25
    Slider (896,109 165x30), variable: PLC_PRG.decomressPress, scale 0..25
    Label (388,236 97x30), "Датчик НД ГРБ"
    Label (389,369 97x30), "Датчик ВД ГРБ"
    Label (353,53 97x30), "Датчик Сжатия"
    Label (779,35 131x30), "Датчик Растяжения"
    Slider (496,29 285x19), variable: PLC_PRG.mowAbsorb, scale 0..36
    BarDisplayImage (621,72 169x31), value: PLC_PRG.rightMowAbsorb, style: BarDisplayImage-Gray, scale format: %.1f, scale 0..15
    BarDisplayImage (476,72 168x31), value: PLC_PRG.leftMowAbsorb, style: BarDisplayImage-Gray, scale format: %.1f, scale 0..15
    Rectangle (623,53 19x61), colour toggle: GVL.defectMowAbsorbSens
    Label (582,13 100x19), "Датчик ХодАмор"
    Line (554,110)
    Ellipse (615,161 9x9)
    Line (603,215)
    Line (613,124) (534,124)
    Line (721,124) (618,124)
    Ellipse (530,120 9x9)
    Ellipse (718,120 9x9)
    Group (606,137 40x19)
        Rectangle (0,1 69x25)
        Line (34,24) (34,0)
    Label (647,138 33x19), "SOL5"
    Line (611,138) (611,122)
    Line (620,137) (620,122)
    Line (723,259) (723,124), colour toggle: GVL.SOL4
    Line (725,257) (619,257), colour toggle: GVL.SOL4
    Line (535,259) (535,124), colour toggle: GVL.SOL3
    Line (614,257) (533,257), colour toggle: GVL.SOL3
    Group (700,175 32x59)
        Rectangle (0,27 56x66)
        Ellipse (3,46 30x30)
        Line (41,94) (41,26)
        Line (8,22) (8,0)
        Line (5,75) (5,53)
        Line (19,46) (19,35)
        Line (19,87) (19,76)
    Group (745,205 40x19)
        Rectangle (0,1 69x25)
        Line (34,24) (34,0)
    Label (763,189 35x19), "SOL11"
    Line (755,177) (722,177), colour toggle: GVL.SOL11
    Line (755,247) (722,247), colour toggle: GVL.SOL11
    Line (753,206) (753,175), colour toggle: GVL.SOL11
    Line (753,249) (753,223), colour toggle: GVL.SOL11
    Ellipse (719,172 9x9)
    Ellipse (718,242 9x9)
    Group (511,176 32x59)
        Rectangle (0,27 56x66)
        Ellipse (3,46 30x30)
        Line (41,94) (41,26)
        Line (8,22) (8,0)
        Line (5,75) (5,53)
        Line (19,46) (19,35)
        Line (19,87) (19,76)
    Group (457,203 40x19)
        Rectangle (0,1 69x25)
        Line (34,24) (34,0)
    Label (448,186 36x19), "SOL10"
    Line (536,179) (488,179), colour toggle: GVL.SOL10
    Line (537,246) (488,246), colour toggle: GVL.SOL10
    Line (490,248) (490,222), colour toggle: GVL.SOL10
    Line (490,205) (490,177), colour toggle: GVL.SOL10
    Group (588,274 60x18)
        Rectangle (0,0 60x18)
        Line (39,17) (39,0)
        Line (19,17) (19,0)
    Line (621,311) (621,291)
    Line (612,552) (612,291), colour toggle: GVL.pumpWork
    Line (621,275) (621,255), colour toggle: GVL.SOL4
    Line (612,275) (612,255), colour toggle: GVL.SOL3
    Line (805,309) (619,309)
    Label (649,273 36x19), "SOL4"
    Label (548,273 36x19), "SOL3"
    Group (692,334 30x41)
        Rectangle (15,0 15x20)
        Line (15,14) (29,14)
        Line (0,40)
        Line (23,31) (23,20)
        Line (23,31) (3,31)
        Line (3,31) (3,8)
    Group (649,388 60x18)
        Rectangle (0,0 60x18)
        Line (39,17) (39,0)
        Line (19,17) (19,0)
    Group (647,433 30x41)
        Rectangle (15,0 15x20)
        Line (15,14) (29,14)
        Line (0,40)
        Line (23,31) (23,20)
        Line (23,31) (3,31)
        Line (3,31) (3,8)
    Line (672,433) (672,406), colour toggle: GVL.SOL1
    Ellipse (530,174 9x9)
    Ellipse (530,241 9x9)
    Ellipse (690,338 9x9)
    Ellipse (645,437 9x9)
    Ellipse (680,436 9x9)
    Group (611,156 10x12)
        Line (9,20) (9,0)
        Line (0,20) (0,0)
    Line (807,166) (609,166)
    Ellipse (597,479 30x30), colour toggle: GVL.pumpWork
    Ellipse (537,480 30x30), "M", colour toggle: GVL.pumpStart
    Line (566,491) (598,491)
    Line (566,500) (598,500)
    Line (805,551) (805,164)
    Ellipse (800,304 9x9)
    Ellipse (800,339 9x9)
    Ellipse (800,437 9x9)
    Ellipse (608,436 9x9)
    Pie (830,570 20x15), colour toggle: GVL.heaterOil
    Line (918,532) (839,532), colour toggle: GVL.heaterOil
    Line (916,586) (837,586), colour toggle: GVL.heaterOil
    Rectangle (916,515 53x87), "БТЭН", colour toggle: GVL.heaterOil
    Group (413,390 100x100)
        Meter360 (0,0 138x134), value: PLC_PRG.hiPres, style: Meter-Meter360-Gray, scale format: %.1f, scale 4..20
        Ellipse (44,45 44x44), colour toggle: GVL.defectHiPresSens
    Line (534,124) (445,124), colour toggle: GVL.SOL3
    Group (352,76 100x100)
        Meter360 (0,0 138x134), value: PLC_PRG.compressPress, style: Meter-Meter360-Gray, scale format: %.1f, scale 4..20
        Ellipse (44,45 44x44), colour toggle: GVL.defectCompressPressSens
    Group (523,371 40x19)
        Rectangle (0,1 69x25)
        Line (34,24) (34,0)
    Label (546,351 36x19), "SOL12"
    Line (531,443) (531,389), colour toggle: GVL.SOL2
    Line (538,371) (538,315), colour toggle: GVL.SOL2
    Line (540,316) (507,316), colour toggle: GVL.SOL2
    Group (415,261 100x100)
        Meter360 (0,0 138x134), value: PLC_PRG.lowPres, style: Meter-Meter360-Gray, scale format: %.1f, scale 4..20
        Ellipse (44,45 44x44), colour toggle: GVL.defectLowPresSens
    Line (814,124) (725,124), colour toggle: GVL.SOL4
    Group (811,60 100x100)
        Meter360 (0,0 138x134), value: PLC_PRG.decomressPress, style: Meter-Meter360-Gray, scale format: %.1f, scale 4..20
        Ellipse (44,45 44x44), colour toggle: GVL.defectDecomressPressSens
    Line (817,561) (817,432)
    Label (819,329 97x30), "Датчик T масла"
    Group (812,358 100x100)
        Meter360 (0,0 100x100), value: PLC_PRG.temperatuteOil, style: Meter-Meter360-Gray, scale format: %.1f, scale 4..20
        Ellipse (32,34 32x33), colour toggle: GVL.defectTemperatuteOilSens
    Pie (831,534 20x15), colour toggle: GVL.heaterOil
    Pie (829,552 20x15), colour toggle: GVL.heaterOil
    Pie (509,570 20x15), colour toggle: GVL.coolerOil
    Line (520,550) (441,550), colour toggle: GVL.coolerOil
    Line (519,568) (440,568), colour toggle: GVL.coolerOil
    Rectangle (356,543 84x31), "Охлаждение", colour toggle: GVL.coolerOil
    Pie (510,534 20x15), colour toggle: GVL.coolerOil
    Pie (508,552 20x15), colour toggle: GVL.coolerOil
    Rectangle (631,481 99x30), "%S", text variable: PLC_PRG.TONPump.ET
    Button (40,26 159x30), "пуск насос", pressed state: GVL.pumpOn
        toggle GVL.pumpOn
    Line (535,124) (535,102), colour toggle: GVL.SOL5
    Line (723,124) (723,102), colour toggle: GVL.SOL5
    Ellipse (631,275 15x15), colour toggle: GVL.SOL4
    Ellipse (590,276 15x15), colour toggle: GVL.SOL3
    Ellipse (546,374 15x15), colour toggle: GVL.SOL2
    Ellipse (629,140 15x15), colour toggle: GVL.SOL5
    Ellipse (607,140 15x15)
    Ellipse (459,206 15x15), colour toggle: GVL.SOL10
    Ellipse (768,207 15x15), colour toggle: GVL.SOL11
    Ellipse (652,389 15x15), colour toggle: GVL.SOL1
    Ellipse (692,390 15x15), colour toggle: GVL.SOL2
    GroupBox (19,126 188x208), "Ручной режим", invisible if: PLC_PRG.onButton
        Button (12,24 165x30), "Высокое давление", invisible if: PLC_PRG.onButton
        Button (12,59 165x30), "Низкое давление", colour toggle: GVL.SOL2
            toggle GVL.SOL2
        Button (12,93 165x30), "Сжатие", colour toggle: GVL.SOL3, invisible if: PLC_PRG.onButton
            toggle GVL.SOL3
        Button (12,127 165x30), "Растяжение", colour toggle: GVL.SOL4
            toggle GVL.SOL4
        Button (11,162 165x30), "Пуск", colour toggle: GVL.SOL5, invisible if: PLC_PRG.onButton
            toggle GVL.SOL5
    GroupBox (19,351 192x208), "Автоматический режим", invisible if: PLC_PRG.onButton
        Button (8,23 176x42), "Нормальная нагрузка", colour toggle: GVL.normalLoadMode, invisible if: PLC_PRG.onButton
            toggle GVL.normalLoadMode
        Button (7,69 176x42), "Открытия клапана", colour toggle: GVL.openMode, invisible if: PLC_PRG.onButton
            toggle GVL.openMode
        Button (8,116 176x42), "Холостой ход", pressed state: GVL.resistanceMode, invisible if: PLC_PRG.onButton
            toggle GVL.resistanceMode
        Button (9,162 176x42), "Скорость закрытия", invisible if: PLC_PRG.onButton
    Label (629,408 36x19), "SOL1"
    Label (694,406 36x19), "SOL2"
    Button (25,65 183x30), "Среднее положение", pressed state: GVL.pumpOn, invisible if: PLC_PRG.onButton
END_VISUALIZATION
